FUNCTION Call_Warehouse

instStackerCrane(XAxisMoving := StackerCraneOneXAxisIsMoving,
				 ZAxisMoving := StackerCraneOneZAxisIsMoving,
				 ActorInstanceIndex := 0,
				 ActorInstanceName := 'Zufuehrung',
				 ForkInPosLeft := Gabel_InPos_Links,
				 ForkInPosMiddle := Gabel_InPos_Mitte,
				 ForkInPosRight := Gabel_InPos_Rechts,
				 OperatingMode := instOperatingMode.StateOperatingMode,
				 HMIInterface := HMI.hmiMachineSectionInterface,
				 LiftFork => StackerCraneOneLiftFork,
				 MoveForkLeft => Gabel_zu_Pos_Links,
				 MoveForkRight => Gabel_zu_Pos_Rechts,
				 TargetPos => StackerCraneOneTargetPos);
				 
(*================ Steps ================*)
IF instOperatingMode.StateOperatingMode.Reset.IsActive THEN
	processStepsLoading := StackerCraneStepsLoading.Waiting;
END_IF

CASE processStepsLoading OF
	StackerCraneStepsLoading.Waiting:
		instStackerCrane.MoveForkToMiddle_ON(TRUE);
		IF instOperatingMode.StateOperatingMode.AutomaticStart.IsActive THEN
			processStepsLoading := StackerCraneStepsLoading.DriveToLoadingPosition;
		END_IF
StackerCraneStepsLoading.DriveToLoadingPosition:
		instStackerCrane.MoveAxesStackerCrane_ON(TRUE, 55);
		IF instStackerCrane.InPositionXAxis AND instStackerCrane.InPositionZAxis   
		AND PartPresentConveyorInfeedStCEnd
		THEN
			InUnloading	:= FALSE;
			processStepsLoading := StackerCraneStepsLoading.ForkUnderLoad;
		END_IF
StackerCraneStepsLoading.ForkUnderLoad:
		InUnloading	:= FALSE;
		instStackerCrane.MoveForkToLeft_ON(TRUE);
		IF Gabel_InPos_Links THEN
			processStepsLoading := StackerCraneStepsLoading.LiftLoadItem;
		END_IF
StackerCraneStepsLoading.LiftLoadItem:
		instStackerCrane.MoveForkToLeft_ON(TRUE);
		instStackerCrane.LiftForkUp(TRUE);
		IF instStackerCrane.InPositionXAxis AND instStackerCrane.InPositionZAxis 
		AND TRUE
		THEN
			processStepsLoading := StackerCraneStepsLoading.ForkToMiddle;
		END_IF
StackerCraneStepsLoading.ForkToMiddle:
		instStackerCrane.MoveForkToMiddle_ON(TRUE);
		IF Gabel_InPos_Mitte AND NOT InUnloading THEN
			processStepsLoading := StackerCraneStepsLoading.DriveToUnloadPrePosition;
		ELSIF Gabel_InPos_Mitte AND InUnloading THEN
			processStepsLoading := StackerCraneStepsLoading.DriveToLoadingPosition;
		END_IF
StackerCraneStepsLoading.DriveToUnloadPrePosition:
		instStackerCrane.MoveAxesStackerCrane_ON(TRUE, 1);
		IF instStackerCrane.InPositionXAxis AND instStackerCrane.InPositionZAxis   
		AND TRUE
		THEN
			processStepsLoading := StackerCraneStepsLoading.ForkInWarehouse;
		END_IF
StackerCraneStepsLoading.ForkInWarehouse:
		instStackerCrane.MoveForkToRight_ON(TRUE);
		IF Gabel_InPos_Rechts THEN
			processStepsLoading := StackerCraneStepsLoading.DriveToUnloadPosition;
		END_IF
StackerCraneStepsLoading.DriveToUnloadPosition:
		instStackerCrane.MoveForkToRight_ON(TRUE);
		instStackerCrane.LowerForkUp(TRUE);
		IF instStackerCrane.InPositionXAxis AND instStackerCrane.InPositionZAxis  
		AND TRUE
		THEN
			InUnloading	:= TRUE;
			processStepsLoading := StackerCraneStepsLoading.ForkToMiddle;
		END_IF
END_CASE

END_FUNCTION

(* stored: Version 1.1.0.1
   POU Call_Warehouse: Id {f6c8f4cf-ee39-4374-8fe6-66362c853c49}, SpecialFunc None *)
